(* IEC 61131-3 sources: std_i2980_v2.06_cp053/Source/IMM/ieccontrol/MoldHeightAdjust1 (part 4) *)

(* ---- ABButtonControl.pu ---- *)
IMPORT_OVER_LISTFILE
 IS_LINKED
, tyPanelButton
, tevPanelButtonRegisterData
, tevPanelButtonRegister
, ABManualButton
, tsDeviceId
, tsPanelButton

END_IMPORT

ALGORITHM_BLOCK ABButtonControl #DUMMY_EDIT_BLOCK

SYSTEM_VAR
 sv_bInitStart : BOOL;
 sv_bDeviceReady : BOOL;
 sv_iPanelMovementSelector : DINT;
 sv_bHMILedAutoAdjust_ledAttr : BYTE;
 sv_bHMILedAutoAdjust : BOOL;
 sv_PanelButtons : tyPanelButton;
 di_ButtonGeneral1 : BOOL;
 di_ButtonGeneral2 : BOOL;
 sv_DeviceId : tsDeviceId;
 di_ButtonStart : BOOL;
 sv_bButtonStart : BOOL;
END_VAR

SYSTEM_OBJECT
 evPanelButtonRegister : tevPanelButtonRegister;
 PU_Task_7 : TASK;
 PU_Task_13 : TASK;
END_OBJECT

VAR
 evPanelButtonRegisterData : tevPanelButtonRegisterData;
 abManualButton : ABManualButton;
 mpbButtonGeneralFwd : REFTO BOOL;
 mpbButtonGeneralBwd : REFTO BOOL;
 mbDIButtonStartLinked : BOOL;
 mbDIButtonGeneral1Linked : BOOL;
 mbDIButtonGeneral2Linked : BOOL;
 mpiPanelMovementSelector : REFTO DINT;
END_VAR

VAR CONSTANT
 cButtonMoveStart : DINT := 1;
END_VAR

POSTUPDATE_ALGORITHM pRegisterButtons ON PU_Task_13 WITH sv_bInitStart

#BEGIN_EDIT_BLOCK
(**************************************** WARNING ********************************************
 *** The KEBA Kemro K2 System including software is not intended for safety control tasks! ***
 ***                       For further information see Comment tab!                        ***
 *********************************************************************************************)

mpbButtonGeneralFwd := EMPTY;
mpbButtonGeneralBwd := EMPTY;

mbDIButtonStartLinked := IS_LINKED(di_ButtonStart);

mbDIButtonGeneral1Linked := IS_LINKED(di_ButtonGeneral1);
mbDIButtonGeneral2Linked := IS_LINKED(di_ButtonGeneral2);

IF (mbDIButtonGeneral1Linked AND mbDIButtonGeneral2Linked) THEN
    mpiPanelMovementSelector := @sv_iPanelMovementSelector;
END_IF;

// register start button
evPanelButtonRegisterData.Button.nPanelButtonType := nPanelButtonMovement;
evPanelButtonRegisterData.Button.iCompId := sv_DeviceId.CompId;
evPanelButtonRegisterData.Button.iIndexId := sv_DeviceId.IndexId;
evPanelButtonRegisterData.Button.iButtonId := cButtonMoveStart;
evPanelButtonRegisterData.Button.pbActionVar1 := @sv_bButtonStart;
evPanelButtonRegisterData.Button.pbActionVar2 := @sv_bButtonStart;
evPanelButtonRegisterData.Button.Optional.pbLedVar := @sv_bHMILedAutoAdjust;
evPanelButtonRegisterData.Button.Optional.piLedVarAttr := @sv_bHMILedAutoAdjust_ledAttr;
SET_EVENT(evPanelButtonRegister, evPanelButtonRegisterData);

;#END_EDIT_BLOCK END_ALGORITHM

POSTUPDATE_ALGORITHM pButtonStart ON PU_Task_7 WITH di_ButtonStart,sv_bButtonStart,mpbButtonGeneralBwd^,mpbButtonGeneralFwd^

VAR
 bButton : BOOL;
END_VAR
#BEGIN_EDIT_BLOCK
(**************************************** WARNING ********************************************
 *** The KEBA Kemro K2 System including software is not intended for safety control tasks! ***
 ***                       For further information see Comment tab!                        ***
 *********************************************************************************************)

// soft panel button
bButton := sv_bButtonStart;

// hw panel button
IF mbDIButtonStartLinked THEN
    bButton := bButton OR di_ButtonStart;
END_IF;

// external panel button
IF CHECK_REF(mpbButtonGeneralBwd^) THEN
    bButton := bButton OR mpbButtonGeneralBwd^;
END_IF;
IF CHECK_REF(mpbButtonGeneralFwd^) THEN
    bButton := bButton OR mpbButtonGeneralFwd^;
END_IF;

abManualButton.aButtonStart(bButtonStart := bButton);

;#END_EDIT_BLOCK END_ALGORITHM

POSTUPDATE_ALGORITHM pMoveSelectorChanged ON PU_Task_7 WITH mpiPanelMovementSelector^

VAR
 Button : tsPanelButton;
END_VAR
#BEGIN_EDIT_BLOCK
(**************************************** WARNING ********************************************
 *** The KEBA Kemro K2 System including software is not intended for safety control tasks! ***
 ***                       For further information see Comment tab!                        ***
 *********************************************************************************************)
mpbButtonGeneralFwd := EMPTY;
mpbButtonGeneralBwd := EMPTY;

IF (NOT sv_bDeviceReady) THEN
    // stop active movements
    abManualButton.aButtonStart(bButtonStart := FALSE);
END_IF;

IF (sv_iPanelMovementSelector > 0) THEN
    Button := sv_PanelButtons[sv_iPanelMovementSelector];
    IF (Button.iCompId = sv_DeviceId.CompId AND
        Button.iIndexId = sv_DeviceId.IndexId) THEN
        IF (Button.iButtonId = cButtonMoveStart) THEN
            mpbButtonGeneralFwd := @di_ButtonGeneral2;
            mpbButtonGeneralBwd := @di_ButtonGeneral1;
        END_IF;
    END_IF;
END_IF;

;#END_EDIT_BLOCK END_ALGORITHM

END_ALGORITHM_BLOCK

#END_OF_IEC_PART

@Puma @IecEditor 6 152 @Pou 25
@@@BEG_Comment@@@

@@@END_Comment@@@

@BEG_Contents

@BEG_Func
@RT(17)FuncTreeContainer
1
@Var @RT(9)IS_LINKED @RT(0) @T @T @DERIVED 0 @F @RT(22)KEBA_STANDARD_FUNCTION @F
@T
@BEG_Attrib
0 @RT(0) @RT(0)
@END_Attrib
1 1 @F @F @F @F

@END_Func

@BEG_Const
@RT(18)ConstTreeContainer
0
@END_Const

@BEG_Export

@BEG_Kind
@ALGORITHM_BLOCK @RT(15)ABButtonControl @STRUCTURED_TEXT
@RT(0) @RT(0) @RT(0)
@END_Kind

@BEG_Dcl
@RT(16)DclTreeContainer
23
@Var @RT(13)sv_bInitStart @RT(0) @T @T @RENAMED 0 @T @T @DT @RT(4)BOOL @RT(0) @T @T @BASIC 0 @F
@F @F
@T
@BEG_Attrib
3 @RT(0) @RT(0) @RT(0)
@END_Attrib
1 8 @F @F @F @F

@Var @RT(15)sv_bDeviceReady @RT(0) @T @T @RENAMED 0 @T @T @DT @RT(4)BOOL @RT(0) @T @T @BASIC 0 @F
@F @F
@T
@BEG_Attrib
3 @RT(0) @RT(0) @RT(0)
@END_Attrib
1 8 @F @F @F @F

@Var @RT(25)sv_iPanelMovementSelector @RT(0) @T @F @DT @RT(4)DINT @RT(0) @T @T @BASIC 0 @F
@F @F
@T
@BEG_Attrib
3 @RT(0) @RT(0) @RT(0)
@END_Attrib
1 8 @F @F @F @F

@Var @RT(28)sv_bHMILedAutoAdjust_ledAttr @RT(0) @T @F @DT @RT(4)BYTE @RT(0) @T @T @BASIC 0 @F
@F @F
@T
@BEG_Attrib
3 @RT(0) @RT(0) @RT(0)
@END_Attrib
1 8 @F @F @F @F

@Var @RT(20)sv_bHMILedAutoAdjust @RT(0) @T @F @DT @RT(4)BOOL @RT(0) @T @T @BASIC 0 @F
@F @F
@T
@BEG_Attrib
3 @RT(0) @RT(0) @RT(0)
@END_Attrib
1 8 @F @F @F @F

@Var @RT(15)sv_PanelButtons @RT(0) @T @T @DERIVED 0 @T @T @DT @RT(13)tyPanelButton @RT(0) @T @T @UNKNOWN 0 @F
@F @F
@T
@BEG_Attrib
3 @RT(0) @RT(0) @RT(0)
@END_Attrib
1 8 @F @F @F @F

@Var @RT(25)evPanelButtonRegisterData @RT(0) @T @T @DERIVED 0 @T @T @DT @RT(26)tevPanelButtonRegisterData @RT(0) @T @T @UNKNOWN 0 @F
@F @F
@T
@BEG_Attrib
3 @RT(0) @RT(0) @RT(0)
@END_Attrib
1 0 @F @F @F @F

@Var @RT(21)evPanelButtonRegister @RT(0) @T @T @DERIVED 0 @T @T @DT @RT(22)tevPanelButtonRegister @RT(0) @T @T @UNKNOWN 0 @F
@F @F
@T
@BEG_Attrib
3 @RT(0) @RT(0) @RT(0)
@END_Attrib
1 7 @F @F @F @F

@Var @RT(14)abManualButton @RT(0) @T @T @DERIVED 0 @T @T @DT @RT(14)ABManualButton @RT(0) @T @T @UNKNOWN 0 @F
@F @F
@T
@BEG_Attrib
3 @RT(0) @RT(0) @RT(0)
@END_Attrib
1 0 @F @F @F @F

@Var @RT(17)di_ButtonGeneral1 @RT(0) @T @F @DT @RT(4)BOOL @RT(0) @T @T @BASIC 0 @F
@F @F
@T
@BEG_Attrib
3 @RT(0) @RT(0) @RT(0)
@END_Attrib
1 8 @F @F @F @F

@Var @RT(17)di_ButtonGeneral2 @RT(0) @T @F @DT @RT(4)BOOL @RT(0) @T @T @BASIC 0 @F
@F @F
@T
@BEG_Attrib
3 @RT(0) @RT(0) @RT(0)
@END_Attrib
1 8 @F @F @F @F

@Var @RT(9)PU_Task_7 @RT(0) @T @F @DT @RT(4)TASK @RT(0) @T @T @BASIC 0 @F
@F @F
@T
@BEG_Attrib
3 @RT(0) @RT(0) @RT(0)
@END_Attrib
1 7 @F @F @F @F

@Var @RT(10)PU_Task_13 @RT(0) @T @T @RENAMED 0 @T @T @DT @RT(4)TASK @RT(0) @T @T @BASIC 0 @F
@F @F
@T
@BEG_Attrib
3 @RT(0) @RT(0) @RT(0)
@END_Attrib
1 7 @F @F @F @F

@Var @RT(11)sv_DeviceId @RT(0) @T @T @DERIVED 0 @T @T @DT @RT(10)tsDeviceId @RT(0) @T @T @UNKNOWN 0 @F
@F @F
@T
@BEG_Attrib
3 @RT(0) @RT(0) @RT(0)
@END_Attrib
1 8 @F @F @F @F

@Var @RT(16)cButtonMoveStart @RT(0) @T @F @DT @RT(4)DINT @RT(0) @T @T @BASIC 0 @F
@F @F
@T
@BEG_Attrib
3 @RT(1)1 @RT(0) @RT(0)
@END_Attrib
1 15 @F @F @F @F

@Var @RT(19)mpbButtonGeneralFwd @RT(0) @T @T @REFTO 0 @T @DT @RT(4)BOOL @RT(0) @T @T @BASIC 0 @F
@F @F
@T
@BEG_Attrib
3 @RT(0) @RT(0) @RT(0)
@END_Attrib
1 0 @F @F @F @F

@Var @RT(19)mpbButtonGeneralBwd @RT(0) @T @T @REFTO 0 @T @DT @RT(4)BOOL @RT(0) @T @T @BASIC 0 @F
@F @F
@T
@BEG_Attrib
3 @RT(0) @RT(0) @RT(0)
@END_Attrib
1 0 @F @F @F @F

@Var @RT(21)mbDIButtonStartLinked @RT(0) @T @F @DT @RT(4)BOOL @RT(0) @T @T @BASIC 0 @F
@F @F
@T
@BEG_Attrib
3 @RT(0) @RT(0) @RT(0)
@END_Attrib
1 0 @F @F @F @F

@Var @RT(24)mbDIButtonGeneral1Linked @RT(0) @T @F @DT @RT(4)BOOL @RT(0) @T @T @BASIC 0 @F
@F @F
@T
@BEG_Attrib
3 @RT(0) @RT(0) @RT(0)
@END_Attrib
1 0 @F @F @F @F

@Var @RT(24)mbDIButtonGeneral2Linked @RT(0) @T @F @DT @RT(4)BOOL @RT(0) @T @T @BASIC 0 @F
@F @F
@T
@BEG_Attrib
3 @RT(0) @RT(0) @RT(0)
@END_Attrib
1 0 @F @F @F @F

@Var @RT(14)di_ButtonStart @RT(0) @T @T @RENAMED 0 @T @T @DT @RT(4)BOOL @RT(0) @T @T @BASIC 0 @F
@F @F
@T
@BEG_Attrib
3 @RT(0) @RT(0) @RT(0)
@END_Attrib
1 8 @F @F @F @F

@Var @RT(15)sv_bButtonStart @RT(0) @T @T @RENAMED 0 @T @T @DT @RT(4)BOOL @RT(0) @T @T @BASIC 0 @F
@F @F
@T
@BEG_Attrib
3 @RT(0) @RT(0) @RT(0)
@END_Attrib
1 8 @F @F @F @F

@Var @RT(24)mpiPanelMovementSelector @RT(0) @T @T @REFTO 0 @T @DT @RT(4)DINT @RT(0) @T @T @BASIC 0 @F
@F @F
@T
@BEG_Attrib
3 @RT(0) @RT(0) @RT(0)
@END_Attrib
1 0 @F @F @F @F

@END_Dcl

@END_Export

@BEG_Body

3

@BEG_Export

@BEG_Algo
@POSTUPDATE_ALGORITHM @RT(16)pRegisterButtons @STRUCTURED_TEXT
@RT(0) @RT(13)sv_bInitStart @RT(10)PU_Task_13 @F @F
@END_Algo

@BEG_Dcl
@RT(16)DclTreeContainer
0
@END_Dcl

@END_Export

@BEG_Export

@BEG_Algo
@POSTUPDATE_ALGORITHM @RT(12)pButtonStart @STRUCTURED_TEXT
@RT(0) @RT(72)di_ButtonStart,sv_bButtonStart,mpbButtonGeneralBwd^,mpbButtonGeneralFwd^ @RT(9)PU_Task_7 @F @F
@END_Algo

@BEG_Dcl
@RT(16)DclTreeContainer
1
@Var @RT(7)bButton @RT(0) @T @F @DT @RT(4)BOOL @RT(0) @T @T @BASIC 0 @F
@F @F
@T
@BEG_Attrib
3 @RT(0) @RT(0) @RT(0)
@END_Attrib
1 0 @F @F @F @F

@END_Dcl

@END_Export

@BEG_Export

@BEG_Algo
@POSTUPDATE_ALGORITHM @RT(20)pMoveSelectorChanged @STRUCTURED_TEXT
@RT(0) @RT(25)mpiPanelMovementSelector^ @RT(9)PU_Task_7 @F @F
@END_Algo

@BEG_Dcl
@RT(16)DclTreeContainer
1
@Var @RT(6)Button @RT(0) @T @T @DERIVED 0 @T @T @DT @RT(13)tsPanelButton @RT(0) @T @T @UNKNOWN 0 @F
@F @F
@T
@BEG_Attrib
3 @RT(0) @RT(0) @RT(0)
@END_Attrib
1 0 @F @F @F @F

@END_Dcl

@END_Export

@BEG_Body
@TL(29)
(**************************************** WARNING ********************************************
 *** The KEBA Kemro K2 System including software is not intended for safety control tasks! ***
 ***                       For further information see Comment tab!                        ***
 *********************************************************************************************)

mpbButtonGeneralFwd := EMPTY;
mpbButtonGeneralBwd := EMPTY;

mbDIButtonStartLinked := IS_LINKED(di_ButtonStart);

mbDIButtonGeneral1Linked := IS_LINKED(di_ButtonGeneral1);
mbDIButtonGeneral2Linked := IS_LINKED(di_ButtonGeneral2);

IF (mbDIButtonGeneral1Linked AND mbDIButtonGeneral2Linked) THEN
    mpiPanelMovementSelector := @sv_iPanelMovementSelector;
END_IF;

// register start button
evPanelButtonRegisterData.Button.nPanelButtonType := nPanelButtonMovement;
evPanelButtonRegisterData.Button.iCompId := sv_DeviceId.CompId;
evPanelButtonRegisterData.Button.iIndexId := sv_DeviceId.IndexId;
evPanelButtonRegisterData.Button.iButtonId := cButtonMoveStart;
evPanelButtonRegisterData.Button.pbActionVar1 := @sv_bButtonStart;
evPanelButtonRegisterData.Button.pbActionVar2 := @sv_bButtonStart;
evPanelButtonRegisterData.Button.Optional.pbLedVar := @sv_bHMILedAutoAdjust;
evPanelButtonRegisterData.Button.Optional.piLedVarAttr := @sv_bHMILedAutoAdjust_ledAttr;
SET_EVENT(evPanelButtonRegister, evPanelButtonRegisterData);

@END_Body

@@@BEG_Comment@@@
@TL(0)

@@@END_Comment@@@

@BEG_Body
@TL(24)
(**************************************** WARNING ********************************************
 *** The KEBA Kemro K2 System including software is not intended for safety control tasks! ***
 ***                       For further information see Comment tab!                        ***
 *********************************************************************************************)

// soft panel button
bButton := sv_bButtonStart;

// hw panel button
IF mbDIButtonStartLinked THEN
    bButton := bButton OR di_ButtonStart;
END_IF;

// external panel button
IF CHECK_REF(mpbButtonGeneralBwd^) THEN
    bButton := bButton OR mpbButtonGeneralBwd^;
END_IF;
IF CHECK_REF(mpbButtonGeneralFwd^) THEN
    bButton := bButton OR mpbButtonGeneralFwd^;
END_IF;

abManualButton.aButtonStart(bButtonStart := bButton);

@END_Body

@@@BEG_Comment@@@
@TL(0)

@@@END_Comment@@@

@BEG_Body
@TL(26)
(**************************************** WARNING ********************************************
 *** The KEBA Kemro K2 System including software is not intended for safety control tasks! ***
 ***                       For further information see Comment tab!                        ***
 *********************************************************************************************)
mpbButtonGeneralFwd := EMPTY;
mpbButtonGeneralBwd := EMPTY;

IF (NOT sv_bDeviceReady) THEN
    // stop active movements
    abManualButton.aButtonStart(bButtonStart := FALSE);
END_IF;

IF (sv_iPanelMovementSelector > 0) THEN
    Button := sv_PanelButtons[sv_iPanelMovementSelector];
    IF (Button.iCompId = sv_DeviceId.CompId AND
        Button.iIndexId = sv_DeviceId.IndexId) THEN
        IF (Button.iButtonId = cButtonMoveStart) THEN
            mpbButtonGeneralFwd := @di_ButtonGeneral2;
            mpbButtonGeneralBwd := @di_ButtonGeneral1;
        END_IF;
    END_IF;
END_IF;

@END_Body

@@@BEG_Comment@@@
@TL(0)

@@@END_Comment@@@
@END_Body

@END_Contents

(* ---- ABCalculateMoldHeightImpulses.pu ---- *)
(*
Calculate number of mold height adjust impulses from clamp force
and clamp force from mold height adjust impulses
*)

IMPORT_OVER_LISTFILE
 KCTRL_Lintab_Light
, KAPPL_LintabData
, KCTRL_Lintab_Param_Light

END_IMPORT

ALGORITHM_BLOCK ABCalculateMoldHeightImpulses #DUMMY_EDIT_BLOCK

VAR
 abKCTRL_Lintab : KCTRL_Lintab_Light;
END_VAR

ALGORITHM aInit

VAR_INPUT
 Lintab : KAPPL_LintabData (* lintab for calculating number of impulses from clamping force *);
END_VAR

VAR_TEMP
 LintabParam : KCTRL_Lintab_Param_Light;
END_VAR
#BEGIN_EDIT_BLOCK
(**************************************** WARNING ********************************************
 *** The KEBA Kemro K2 System including software is not intended for safety control tasks! ***
 ***                       For further information see Comment tab!                        ***
 *********************************************************************************************)

LintabParam.LintabPoints := Lintab.LintabPoints;
LintabParam.Mode.bLinearExtrapolation := TRUE;
LintabParam.Mode.bSetNegativeValuesToZero := TRUE;
LintabParam.Mode.bZeroExtrapolation := FALSE;
abKCTRL_Lintab.Par(Param := LintabParam);
abKCTRL_Lintab.Init();

;#END_EDIT_BLOCK END_ALGORITHM

ALGORITHM aCalc

VAR_INPUT
 rForce : REAL (* wanted clamping force *);
END_VAR

VAR_OUTPUT
 iImpulses : DINT (* number of impulses needed for given force *);
END_VAR
#BEGIN_EDIT_BLOCK
(**************************************** WARNING ********************************************
 *** The KEBA Kemro K2 System including software is not intended for safety control tasks! ***
 ***                       For further information see Comment tab!                        ***
 *********************************************************************************************)

//calculate number of impulses from clamping force lintab

abKCTRL_Lintab.CalculateInv(rY := rForce);
iImpulses := REAL_TO_DINT(abKCTRL_Lintab.CalculateInv.rX);

;#END_EDIT_BLOCK END_ALGORITHM

ALGORITHM aCalcInv

VAR_INPUT
 iImpulses : DINT (* number of impulses *);
END_VAR

VAR_OUTPUT
 rForce : REAL (* force from given number of impulses *);
END_VAR
#BEGIN_EDIT_BLOCK
(**************************************** WARNING ********************************************
 *** The KEBA Kemro K2 System including software is not intended for safety control tasks! ***
 ***                       For further information see Comment tab!                        ***
 *********************************************************************************************)

abKCTRL_Lintab.Calculate(rX := DINT_TO_REAL(iImpulses));
rForce := abKCTRL_Lintab.Calculate.rY;

;#END_EDIT_BLOCK END_ALGORITHM

END_ALGORITHM_BLOCK

#END_OF_IEC_PART

@Puma @IecEditor 6 30 @Pou 25
@@@BEG_Comment@@@
Calculate number of mold height adjust impulses from clamp force
and clamp force from mold height adjust impulses
@@@END_Comment@@@

@BEG_Contents

@BEG_Func
@RT(17)FuncTreeContainer
0
@END_Func

@BEG_Const
@RT(18)ConstTreeContainer
0
@END_Const

@BEG_Export

@BEG_Kind
@ALGORITHM_BLOCK @RT(29)ABCalculateMoldHeightImpulses @STRUCTURED_TEXT
@RT(0) @RT(0) @RT(0)
@END_Kind

@BEG_Dcl
@RT(16)DclTreeContainer
1
@Var @RT(14)abKCTRL_Lintab @RT(0) @T @T @DERIVED 0 @T @T @DT @RT(18)KCTRL_Lintab_Light @RT(0) @T @T @UNKNOWN 0 @F
@F @F
@T
@BEG_Attrib
3 @RT(0) @RT(0) @RT(0)
@END_Attrib
1 0 @F @F @F @F

@END_Dcl

@END_Export

@BEG_Body

3

@BEG_Export

@BEG_Algo
@ALGORITHM @RT(5)aInit @STRUCTURED_TEXT
@RT(0) @RT(0) @RT(0) @F @F
@END_Algo

@BEG_Dcl
@RT(16)DclTreeContainer
2
@Var @RT(6)Lintab @RT(0) @T @T @DERIVED 0 @T @T @DT @RT(16)KAPPL_LintabData @RT(0) @T @T @UNKNOWN 0 @F
@F @F
@T
@BEG_Attrib
3 @RT(0) @RT(61)lintab for calculating number of impulses from clamping force @RT(0)
@END_Attrib
1 1 @F @F @F @F

@Var @RT(11)LintabParam @RT(0) @T @T @DERIVED 0 @T @T @DT @RT(24)KCTRL_Lintab_Param_Light @RT(0) @T @T @UNKNOWN 0 @F
@F @F
@T
@BEG_Attrib
3 @RT(0) @RT(0) @RT(0)
@END_Attrib
1 4 @F @F @F @F

@END_Dcl

@END_Export

@BEG_Export

@BEG_Algo
@ALGORITHM @RT(5)aCalc @STRUCTURED_TEXT
@RT(0) @RT(0) @RT(0) @F @F
@END_Algo

@BEG_Dcl
@RT(16)DclTreeContainer
2
@Var @RT(6)rForce @RT(0) @T @F @DT @RT(4)REAL @RT(0) @T @T @BASIC 0 @F
@F @F
@T
@BEG_Attrib
3 @RT(0) @RT(21)wanted clamping force @RT(0)
@END_Attrib
1 1 @F @F @F @F

@Var @RT(9)iImpulses @RT(0) @T @F @DT @RT(4)DINT @RT(0) @T @T @BASIC 0 @F
@F @F
@T
@BEG_Attrib
3 @RT(0) @RT(41)number of impulses needed for given force @RT(0)
@END_Attrib
1 3 @F @F @F @F

@END_Dcl

@END_Export

@BEG_Export

@BEG_Algo
@ALGORITHM @RT(8)aCalcInv @STRUCTURED_TEXT
@RT(0) @RT(0) @RT(0) @F @F
@END_Algo

@BEG_Dcl
@RT(16)DclTreeContainer
2
@Var @RT(9)iImpulses @RT(0) @T @F @DT @RT(4)DINT @RT(0) @T @T @BASIC 0 @F
@F @F
@T
@BEG_Attrib
3 @RT(0) @RT(18)number of impulses @RT(0)
@END_Attrib
1 1 @F @F @F @F

@Var @RT(6)rForce @RT(0) @T @F @DT @RT(4)REAL @RT(0) @T @T @BASIC 0 @F
@F @F
@T
@BEG_Attrib
3 @RT(0) @RT(35)force from given number of impulses @RT(0)
@END_Attrib
1 3 @F @F @F @F

@END_Dcl

@END_Export

@BEG_Body
@TL(12)
(**************************************** WARNING ********************************************
 *** The KEBA Kemro K2 System including software is not intended for safety control tasks! ***
 ***                       For further information see Comment tab!                        ***
 *********************************************************************************************)

LintabParam.LintabPoints := Lintab.LintabPoints;
LintabParam.Mode.bLinearExtrapolation := TRUE;
LintabParam.Mode.bSetNegativeValuesToZero := TRUE;
LintabParam.Mode.bZeroExtrapolation := FALSE;
abKCTRL_Lintab.Par(Param := LintabParam);
abKCTRL_Lintab.Init();

@END_Body

@@@BEG_Comment@@@
@TL(0)

@@@END_Comment@@@

@BEG_Body
@TL(11)
(**************************************** WARNING ********************************************
 *** The KEBA Kemro K2 System including software is not intended for safety control tasks! ***
 ***                       For further information see Comment tab!                        ***
 *********************************************************************************************)

//calculate number of impulses from clamping force lintab

abKCTRL_Lintab.CalculateInv(rY := rForce);
iImpulses := REAL_TO_DINT(abKCTRL_Lintab.CalculateInv.rX);

@END_Body

@@@BEG_Comment@@@
@TL(0)

@@@END_Comment@@@

@BEG_Body
@TL(9)
(**************************************** WARNING ********************************************
 *** The KEBA Kemro K2 System including software is not intended for safety control tasks! ***
 ***                       For further information see Comment tab!                        ***
 *********************************************************************************************)

abKCTRL_Lintab.Calculate(rX := DINT_TO_REAL(iImpulses));
rForce := abKCTRL_Lintab.Calculate.rY;

@END_Body

@@@BEG_Comment@@@
@TL(0)

@@@END_Comment@@@
@END_Body

@END_Contents

(* ---- ABCalculateMoldHeightMm.pu ---- *)
(*
Calculate number of mold height adjust impulses from clamp force
and clamp force from mold height adjust impulses
*)

IMPORT_OVER_LISTFILE
 KCTRL_Lintab_Light
, KAPPL_LintabData
, KCTRL_Lintab_Param_Light

END_IMPORT

ALGORITHM_BLOCK ABCalculateMoldHeightMm #DUMMY_EDIT_BLOCK

VAR
 abKCTRL_Lintab_ClampF : KCTRL_Lintab_Light;
 abKCTRL_Lintab_ToggleLever : KCTRL_Lintab_Light;
END_VAR

ALGORITHM aInit

VAR_INPUT
 LintabClampF : KAPPL_LintabData (* lintab for calculating mold open length from clamping force *);
 LintabToggleLever : KAPPL_LintabData (* lintab for calculating mold open length from clamping force *);
END_VAR

VAR_TEMP
 LintabParam : KCTRL_Lintab_Param_Light;
END_VAR
#BEGIN_EDIT_BLOCK
(**************************************** WARNING ********************************************
 *** The KEBA Kemro K2 System including software is not intended for safety control tasks! ***
 ***                       For further information see Comment tab!                        ***
 *********************************************************************************************)

LintabParam.Mode.bLinearExtrapolation := TRUE;
LintabParam.Mode.bSetNegativeValuesToZero := TRUE;
LintabParam.Mode.bZeroExtrapolation := FALSE;

LintabParam.LintabPoints := LintabClampF.LintabPoints;
abKCTRL_Lintab_ClampF.Par(Param := LintabParam);
abKCTRL_Lintab_ClampF.Init();

LintabParam.LintabPoints := LintabToggleLever.LintabPoints;
abKCTRL_Lintab_ToggleLever.Par(Param := LintabParam);
abKCTRL_Lintab_ToggleLever.Init();

;#END_EDIT_BLOCK END_ALGORITHM

ALGORITHM aCalc

VAR_INPUT
 rForce : REAL (* wanted clamping force *);
END_VAR

VAR_OUTPUT
 rToggleLeverPos : REAL (* new mold offset for given force *);
 rMoldPos : REAL;
END_VAR
#BEGIN_EDIT_BLOCK
(**************************************** WARNING ********************************************
 *** The KEBA Kemro K2 System including software is not intended for safety control tasks! ***
 ***                       For further information see Comment tab!                        ***
 *********************************************************************************************)

//length mold has to open from clamping force lintab

abKCTRL_Lintab_ClampF.CalculateInv(rY := rForce);
rMoldPos := abKCTRL_Lintab_ClampF.CalculateInv.rX;

//getting eqivalent toggleleverpos
abKCTRL_Lintab_ToggleLever.CalculateInv(rY := rMoldPos);
rToggleLeverPos := abKCTRL_Lintab_ToggleLever.CalculateInv.rX;

;#END_EDIT_BLOCK END_ALGORITHM

ALGORITHM aCalcInv

// VAR_INPUT
 // rMoldPos : REAL (* mold position *);
// END_VAR

// VAR_OUTPUT
 // rForce : REAL (* force from given number of impulses *);
// END_VAR
#BEGIN_EDIT_BLOCK
(**************************************** WARNING ********************************************
 *** The KEBA Kemro K2 System including software is not intended for safety control tasks! ***
 ***                       For further information see Comment tab!                        ***
 *********************************************************************************************)

//abKCTRL_Lintab.Calculate(rX := rMoldPos);
//rForce := abKCTRL_Lintab.Calculate.rY;

;#END_EDIT_BLOCK END_ALGORITHM

END_ALGORITHM_BLOCK

#END_OF_IEC_PART

@Puma @IecEditor 6 68 @Pou 25
@@@BEG_Comment@@@
Calculate number of mold height adjust impulses from clamp force
and clamp force from mold height adjust impulses
@@@END_Comment@@@

@BEG_Contents

@BEG_Func
@RT(17)FuncTreeContainer
0
@END_Func

@BEG_Const
@RT(18)ConstTreeContainer
0
@END_Const

@BEG_Export

@BEG_Kind
@ALGORITHM_BLOCK @RT(23)ABCalculateMoldHeightMm @STRUCTURED_TEXT
@RT(0) @RT(0) @RT(0)
@END_Kind

@BEG_Dcl
@RT(16)DclTreeContainer
2
@Var @RT(21)abKCTRL_Lintab_ClampF @RT(0) @T @T @DERIVED 0 @T @T @DT @RT(18)KCTRL_Lintab_Light @RT(0) @T @T @UNKNOWN 0 @F
@F @F
@T
@BEG_Attrib
3 @RT(0) @RT(0) @RT(0)
@END_Attrib
1 0 @F @F @F @F

@Var @RT(26)abKCTRL_Lintab_ToggleLever @RT(0) @T @T @DERIVED 0 @T @T @DT @RT(18)KCTRL_Lintab_Light @RT(0) @T @T @UNKNOWN 0 @F
@F @F
@T
@BEG_Attrib
3 @RT(0) @RT(0) @RT(0)
@END_Attrib
1 0 @F @F @F @F

@END_Dcl

@END_Export

@BEG_Body

3

@BEG_Export

@BEG_Algo
@ALGORITHM @RT(5)aInit @STRUCTURED_TEXT
@RT(0) @RT(0) @RT(0) @F @F
@END_Algo

@BEG_Dcl
@RT(16)DclTreeContainer
3
@Var @RT(12)LintabClampF @RT(0) @T @T @DERIVED 0 @T @T @DT @RT(16)KAPPL_LintabData @RT(0) @T @T @UNKNOWN 0 @F
@F @F
@T
@BEG_Attrib
3 @RT(0) @RT(59)lintab for calculating mold open length from clamping force @RT(0)
@END_Attrib
1 1 @F @F @F @F

@Var @RT(17)LintabToggleLever @RT(0) @T @T @DERIVED 0 @T @T @DT @RT(16)KAPPL_LintabData @RT(0) @T @T @UNKNOWN 0 @F
@F @F
@T
@BEG_Attrib
3 @RT(0) @RT(59)lintab for calculating mold open length from clamping force @RT(0)
@END_Attrib
1 1 @F @F @F @F

@Var @RT(11)LintabParam @RT(0) @T @T @DERIVED 0 @T @T @DT @RT(24)KCTRL_Lintab_Param_Light @RT(0) @T @T @UNKNOWN 0 @F
@F @F
@T
@BEG_Attrib
3 @RT(0) @RT(0) @RT(0)
@END_Attrib
1 4 @F @F @F @F

@END_Dcl

@END_Export

@BEG_Export

@BEG_Algo
@ALGORITHM @RT(5)aCalc @STRUCTURED_TEXT
@RT(0) @RT(0) @RT(0) @F @F
@END_Algo

@BEG_Dcl
@RT(16)DclTreeContainer
3
@Var @RT(6)rForce @RT(0) @T @F @DT @RT(4)REAL @RT(0) @T @T @BASIC 0 @F
@F @F
@T
@BEG_Attrib
3 @RT(0) @RT(21)wanted clamping force @RT(0)
@END_Attrib
1 1 @F @F @F @F

@Var @RT(15)rToggleLeverPos @RT(0) @T @F @DT @RT(4)REAL @RT(0) @T @T @BASIC 0 @F
@F @F
@T
@BEG_Attrib
3 @RT(0) @RT(31)new mold offset for given force @RT(0)
@END_Attrib
1 3 @F @F @F @F

@Var @RT(8)rMoldPos @RT(0) @T @F @DT @RT(4)REAL @RT(0) @T @T @BASIC 0 @F
@F @F
@T
@BEG_Attrib
3 @RT(0) @RT(0) @RT(0)
@END_Attrib
1 3 @F @F @F @F

@END_Dcl

@END_Export

@BEG_Export

@BEG_Algo
@ALGORITHM @RT(8)aCalcInv @STRUCTURED_TEXT
@RT(0) @RT(0) @RT(0) @F @F
@END_Algo

@BEG_Dcl
@RT(16)DclTreeContainer
2
@Var @RT(8)rMoldPos @RT(0) @T @F @DT @RT(4)REAL @RT(0) @T @T @BASIC 0 @F
@F @T
@T
@BEG_Attrib
3 @RT(0) @RT(13)mold position @RT(0)
@END_Attrib
1 1 @F @F @F @F

@Var @RT(6)rForce @RT(0) @T @F @DT @RT(4)REAL @RT(0) @T @T @BASIC 0 @F
@F @T
@T
@BEG_Attrib
3 @RT(0) @RT(35)force from given number of impulses @RT(0)
@END_Attrib
1 3 @F @F @F @F

@END_Dcl

@END_Export

@BEG_Body
@TL(18)
(**************************************** WARNING ********************************************
 *** The KEBA Kemro K2 System including software is not intended for safety control tasks! ***
 ***                       For further information see Comment tab!                        ***
 *********************************************************************************************)

LintabParam.Mode.bLinearExtrapolation := TRUE;
LintabParam.Mode.bSetNegativeValuesToZero := TRUE;
LintabParam.Mode.bZeroExtrapolation := FALSE;

LintabParam.LintabPoints := LintabClampF.LintabPoints;
abKCTRL_Lintab_ClampF.Par(Param := LintabParam);
abKCTRL_Lintab_ClampF.Init();

LintabParam.LintabPoints := LintabToggleLever.LintabPoints;
abKCTRL_Lintab_ToggleLever.Par(Param := LintabParam);
abKCTRL_Lintab_ToggleLever.Init();

@END_Body

@@@BEG_Comment@@@
@TL(0)

@@@END_Comment@@@

@BEG_Body
@TL(16)
(**************************************** WARNING ********************************************
 *** The KEBA Kemro K2 System including software is not intended for safety control tasks! ***
 ***                       For further information see Comment tab!                        ***
 *********************************************************************************************)

//length mold has to open from clamping force lintab

abKCTRL_Lintab_ClampF.CalculateInv(rY := rForce);
rMoldPos := abKCTRL_Lintab_ClampF.CalculateInv.rX;

//getting eqivalent toggleleverpos
abKCTRL_Lintab_ToggleLever.CalculateInv(rY := rMoldPos);
rToggleLeverPos := abKCTRL_Lintab_ToggleLever.CalculateInv.rX;

@END_Body

@@@BEG_Comment@@@
@TL(0)

@@@END_Comment@@@

@BEG_Body
@TL(9)
(**************************************** WARNING ********************************************
 *** The KEBA Kemro K2 System including software is not intended for safety control tasks! ***
 ***                       For further information see Comment tab!                        ***
 *********************************************************************************************)

//abKCTRL_Lintab.Calculate(rX := rMoldPos);
//rForce := abKCTRL_Lintab.Calculate.rY;

@END_Body

@@@BEG_Comment@@@
@TL(0)

@@@END_Comment@@@
@END_Body

@END_Contents

(* ---- ABManualButton.pu ---- *)
(*
@h    ! WARNING !
@h    The Kemro K2 system (including software) only meets category B according to EN 954-1,
@h    thus it is not intended for usage in safety-relevant control applications in the field
@h    of personal safety (e.g. emergency stop).
@h    To implement potentially necessary safety-relevant control tasks, always use additional
@h    external safety devices that are intended for the particular purpose, and meet the necessary
@h    functional safety.
@h    For further information see EN 954-1 (EN ISO 13849-1) and/or the K2-x00 user manual, chapter
@h    "CE conformity, directives and standards".

This algo block starts the automatic mold height adjustment by calling the
system.FBManualButton with the correct parameters corresponding to a pressed Panel Button.
*)

IMPORT_OVER_LISTFILE
 SET_ALARM
, nSetup
, cCompMold
, cCompMoldHeight
, tevStartedStopped
, tsMoveData
, tnOperationMode
, tsDeviceId
, FBManualButtonKeep
, tsAlarm
, FBCheckReady
, FBCheckPosReached
, tevStartedStoppedData

END_IMPORT

ALGORITHM_BLOCK ABManualButton #DUMMY_EDIT_BLOCK

SYSTEM_VAR
 sv_MoveMoldHeightAuto : tsMoveData;
 sv_bAutoMoldHeightAdjustActive : BOOL (* is TRUE when auto mold height adjust is acitve *);
 sv_bLedAutoAdjust_ledAttr : BYTE (* LED Attribute *);
 sv_bHMILedAutoAdjust : BOOL;
 sv_bHMILedAutoAdjust_ledAttr : BYTE (* LED Attribute *);
 sv_bLedAutoAdjust : BOOL;
 sv_bInitStart : BOOL;
 sv_OperationMode : tnOperationMode;
 sv_bInitDone : BOOL;
 sv_DeviceId : tsDeviceId;
 sv_bMoldHeightAutoAdjHMI : BOOL (* hmi can start/stop automh adjust with this SV *);
 sv_bDeviceReady : BOOL;
END_VAR

SYSTEM_OBJECT
 PU_Task_7 : TASK;
 EV_Task_7 : TASK;
 erSetupModeRequiredForAdjust : ALARM;
 evStartedStopped : tevStartedStopped;
END_OBJECT

VAR_EXTERNAL
 g_b2Platen : BOOL;
END_VAR

VAR
 fbManualButton : FBManualButtonKeep;
 mpbMoldReady : REFTO BOOL;
 mpbMoldHeightReady : REFTO BOOL;
 mpbNutsOpen : REFTO BOOL;
 mAlarmNutsNotOpen : tsAlarm;
END_VAR

(*
This algo starts the mold height automatic adjustment by calling the
system.FBManualButton with the correct parameters when the di_ButtonIn is
pressed. (post update).
*)

ALGORITHM aStartStop

VAR_INPUT
 bStart : BOOL;
END_VAR
#BEGIN_EDIT_BLOCK
(**************************************** WARNING ********************************************
 *** The KEBA Kemro K2 System including software is not intended for safety control tasks! ***
 ***                       For further information see Comment tab!                        ***
 *********************************************************************************************)

IF (bStart AND (sv_OperationMode <> nSetup)) THEN
   //ignore button if operation mode is not setup
   SET_ALARM(Name := erSetupModeRequiredForAdjust,
            SubID1 := sv_DeviceId.CompId);
   sv_bMoldHeightAutoAdjHMI := FALSE;
   RETURN;
END_IF;

IF bStart AND g_b2Platen THEN
   //ignore button if lock nuts are not open
   IF NOT mpbNutsOpen^ THEN
      SET_ALARM(Name := mAlarmNutsNotOpen.AlarmId);
      sv_bMoldHeightAutoAdjHMI := FALSE;
      RETURN;
   END_IF;
END_IF;

IF (bStart AND sv_bDeviceReady) THEN
   IF (mpbMoldReady <> EMPTY AND NOT mpbMoldReady^) OR (mpbMoldHeightReady <> EMPTY AND NOT mpbMoldHeightReady^) THEN
      // auto adjust should be started and mold movement or mold adjust movement acitve
      // -> ignore manual button
      RETURN;
   END_IF;
END_IF;

(*@ MoldHeightAdjustN.ABManualButton.pButtonStart.Call the fbManualButton using the sv_MoveMoldHeightAuto parameters *)
IF (bStart AND sv_bDeviceReady) OR ((NOT bStart) AND (NOT sv_bDeviceReady)) THEN
   fbManualButton(bButton := TRUE, MoveId := sv_MoveMoldHeightAuto.MoveId, MoveDir := sv_MoveMoldHeightAuto.MoveDir);
END_IF;

;#END_EDIT_BLOCK END_ALGORITHM

(*
This algo starts the mold height automatic adjustment by calling the
system.FBManualButton with the correct parameters when the di_ButtonIn is
pressed. (post update).
*)

ALGORITHM aButtonStart

VAR_INPUT
 bButtonStart : BOOL;
END_VAR
#BEGIN_EDIT_BLOCK
(**************************************** WARNING ********************************************
 *** The KEBA Kemro K2 System including software is not intended for safety control tasks! ***
 ***                       For further information see Comment tab!                        ***
 *********************************************************************************************)

IF bButtonStart THEN
    sv_bMoldHeightAutoAdjHMI := NOT sv_bMoldHeightAutoAdjHMI;
END_IF;

;#END_EDIT_BLOCK END_ALGORITHM

(*
This algo starts the mold height automatic adjustment by calling the
system.FBManualButton with the correct parameters when the di_ButtonIn is
pressed. (post update).
*)

POSTUPDATE_ALGORITHM pHMIStart ON PU_Task_7 WITH sv_bMoldHeightAutoAdjHMI

#BEGIN_EDIT_BLOCK
(**************************************** WARNING ********************************************
 *** The KEBA Kemro K2 System including software is not intended for safety control tasks! ***
 ***                       For further information see Comment tab!                        ***
 *********************************************************************************************)

IF (sv_bMoldHeightAutoAdjHMI AND sv_bDeviceReady) THEN
    aStartStop(TRUE);
ELSIF ((NOT sv_bMoldHeightAutoAdjHMI) AND (NOT sv_bDeviceReady)) THEN
    aStartStop(FALSE);
END_IF;

;#END_EDIT_BLOCK END_ALGORITHM

POSTUPDATE_ALGORITHM pLedControl ON PU_Task_7 WITH sv_bAutoMoldHeightAdjustActive,sv_bInitStart

VAR
 bInitDone : BOOL;
 mbLedAutoAdjustExists : BOOL := FALSE;
END_VAR
#BEGIN_EDIT_BLOCK
(**************************************** WARNING ********************************************
 *** The KEBA Kemro K2 System including software is not intended for safety control tasks! ***
 ***                       For further information see Comment tab!                        ***
 *********************************************************************************************)

IF NOT bInitDone THEN
    sv_bHMILedAutoAdjust_ledAttr := 16#3;
    IF IS_LINKED(sv_bLedAutoAdjust) AND IS_LINKED(sv_bLedAutoAdjust_ledAttr) THEN
        sv_bLedAutoAdjust_ledAttr := sv_bHMILedAutoAdjust_ledAttr;
        mbLedAutoAdjustExists := TRUE;
    ELSE
        mbLedAutoAdjustExists := FALSE;
    END_IF;

    bInitDone := TRUE;
END_IF;

sv_bHMILedAutoAdjust := sv_bAutoMoldHeightAdjustActive;
IF mbLedAutoAdjustExists THEN
    sv_bLedAutoAdjust := sv_bHMILedAutoAdjust;
END_IF;

;#END_EDIT_BLOCK END_ALGORITHM

POSTUPDATE_ALGORITHM pInitDone ON PU_Task_7(10) WITH sv_bInitDone

VAR
 fbCheckReady : FBCheckReady;
 DeviceId : tsDeviceId;
 fbCheckPosReached : FBCheckPosReached;
END_VAR
#BEGIN_EDIT_BLOCK
(**************************************** WARNING ********************************************
 *** The KEBA Kemro K2 System including software is not intended for safety control tasks! ***
 ***                       For further information see Comment tab!                        ***
 *********************************************************************************************)

//get reference to ready flag of mold function unit
DeviceId.CompId := cCompMold;
DeviceId.IndexId := sv_DeviceId.IndexId;
fbCheckReady(DeviceId := DeviceId);
mpbMoldReady := fbCheckReady.pbReady;

//get reference to ready flag of mold adjust function unit
DeviceId.CompId := cCompMoldHeight;
DeviceId.IndexId := sv_DeviceId.IndexId;
fbCheckReady(DeviceId := DeviceId);
mpbMoldHeightReady := fbCheckReady.pbReady;

//get reference to mold nut open movement and save according alarm
IF g_b2Platen THEN
   DeviceId.CompId := cCompMoldNuts;
   DeviceId.IndexId := sv_DeviceId.IndexId;
   fbCheckPosReached(DeviceId := DeviceId,
                     MoveDir := cMoveOpen,
                     MoveId := cMoveOpen);

   mpbNutsOpen := fbCheckPosReached.pbPosReached;
   mAlarmNutsNotOpen := fbCheckPosReached.Alarm;
END_IF;

;#END_EDIT_BLOCK END_ALGORITHM

(*
Manage list and count of currently started movments
in sv_StartedMovements when receiving evStartedStopped events
*)

EVENT_ALGORITHM evaStartedStopped ON EV_Task_7 WITH evStartedStopped

VAR_INPUT
 evStartedStoppedData : tevStartedStoppedData;
END_VAR
#BEGIN_EDIT_BLOCK
(**************************************** WARNING ********************************************
 *** The KEBA Kemro K2 System including software is not intended for safety control tasks! ***
 ***                       For further information see Comment tab!                        ***
 *********************************************************************************************)

IF evStartedStoppedData.MoveId = cMoldHeightAutomatic AND evStartedStoppedData.DeviceId = sv_DeviceId THEN
   IF evStartedStoppedData.State = nStopped OR evStartedStoppedData.State = nStartNotAllowed THEN
      //reset flag when movement in state nStopped OR nStartNotAllowed
      //we can not use a POSTUPDATE on sv_bDeviceReady and check for TRUE because the movement might be locked
      // -> sv_bDeviceReady never goes FALSE -> no POSTUPDATE is executed
      //also we can not use evMovementState because this one is not set by mold height adjust admin
      sv_bMoldHeightAutoAdjHMI := FALSE;
   END_IF;
END_IF;

;#END_EDIT_BLOCK END_ALGORITHM

END_ALGORITHM_BLOCK

#END_OF_IEC_PART

@Puma @IecEditor 6 114 @Pou 25
@@@BEG_Comment@@@
@h    ! WARNING !
@h    The Kemro K2 system (including software) only meets category B according to EN 954-1,
@h    thus it is not intended for usage in safety-relevant control applications in the field
@h    of personal safety (e.g. emergency stop).
@h    To implement potentially necessary safety-relevant control tasks, always use additional
@h    external safety devices that are intended for the particular purpose, and meet the necessary
@h    functional safety.
@h    For further information see EN 954-1 (EN ISO 13849-1) and/or the K2-x00 user manual, chapter
@h    "CE conformity, directives and standards".

This algo block starts the automatic mold height adjustment by calling the
system.FBManualButton with the correct parameters corresponding to a pressed Panel Button.
@@@END_Comment@@@

@BEG_Contents

@BEG_Func
@RT(17)FuncTreeContainer
1
@Var @RT(9)SET_ALARM @RT(0) @T @T @DERIVED 0 @F @RT(23)KEBA_STANDARD_PROCEDURE @F
@T
@BEG_Attrib
0 @RT(0) @RT(0)
@END_Attrib
1 1 @F @F @F @F

@END_Func

@BEG_Const
@RT(18)ConstTreeContainer
3
@Var @RT(6)nSetup @RT(0) @T @T @DERIVED 0 @F @RT(15)tnOperationMode @F
@T
@BEG_Attrib
0 @RT(1)0 @RT(36)Setup mode only for service engineer
@END_Attrib
1 1 @F @F @F @F

@Var @RT(9)cCompMold @RT(0) @T @F @DT @RT(4)DINT @RT(0) @T @T @BASIC 0 @F
@F @F
@T
@BEG_Attrib
0 @RT(3)101 @RT(14)Component Mold
@END_Attrib
1 1 @F @F @F @F

@Var @RT(15)cCompMoldHeight @RT(0) @T @F @DT @RT(4)DINT @RT(0) @T @T @BASIC 0 @F
@F @F
@T
@BEG_Attrib
0 @RT(3)124 @RT(21)Component Mold Height
@END_Attrib
1 1 @F @F @F @F

@END_Const

@BEG_Export

@BEG_Kind
@ALGORITHM_BLOCK @RT(14)ABManualButton @STRUCTURED_TEXT
@RT(0) @RT(0) @RT(0)
@END_Kind

@BEG_Dcl
@RT(16)DclTreeContainer
22
@Var @RT(9)PU_Task_7 @RT(0) @T @F @DT @RT(4)TASK @RT(0) @T @T @BASIC 0 @F
@F @F
@T
@BEG_Attrib
3 @RT(0) @RT(0) @RT(0)
@END_Attrib
1 7 @F @F @F @F

@Var @RT(9)EV_Task_7 @RT(0) @T @F @DT @RT(4)TASK @RT(0) @T @T @BASIC 0 @F
@F @F
@T
@BEG_Attrib
3 @RT(0) @RT(0) @RT(0)
@END_Attrib
1 7 @F @F @F @F

@Var @RT(28)erSetupModeRequiredForAdjust @RT(0) @T @F @DT @RT(5)ALARM @RT(0) @T @T @BASIC 0 @F
@F @F
@T
@BEG_Attrib
3 @RT(0) @RT(0) @RT(0)
@END_Attrib
1 7 @F @F @F @F

@Var @RT(16)evStartedStopped @RT(0) @T @T @DERIVED 0 @T @T @DT @RT(17)tevStartedStopped @RT(0) @T @T @UNKNOWN 0 @F
@F @F
@T
@BEG_Attrib
3 @RT(0) @RT(0) @RT(0)
@END_Attrib
1 7 @F @F @F @F

@Var @RT(21)sv_MoveMoldHeightAuto @RT(0) @T @T @DERIVED 0 @T @T @DT @RT(10)tsMoveData @RT(0) @T @T @UNKNOWN 0 @F
@F @F
@T
@BEG_Attrib
3 @RT(0) @RT(0) @RT(0)
@END_Attrib
1 8 @F @F @F @F

@Var @RT(30)sv_bAutoMoldHeightAdjustActive @RT(0) @T @F @DT @RT(4)BOOL @RT(0) @T @T @BASIC 0 @F
@F @F
@T
@BEG_Attrib
3 @RT(0) @RT(46)is TRUE when auto mold height adjust is acitve @RT(0)
@END_Attrib
1 8 @F @F @F @F

@Var @RT(25)sv_bLedAutoAdjust_ledAttr @RT(0) @T @F @DT @RT(4)BYTE @RT(0) @T @T @BASIC 0 @F
@F @F
@T
@BEG_Attrib
3 @RT(0) @RT(13)LED Attribute @RT(0)
@END_Attrib
1 8 @F @F @F @F

@Var @RT(20)sv_bHMILedAutoAdjust @RT(0) @T @F @DT @RT(4)BOOL @RT(0) @T @T @BASIC 0 @F
@F @F
@T
@BEG_Attrib
3 @RT(0) @RT(0) @RT(0)
@END_Attrib
1 8 @F @F @F @F

@Var @RT(28)sv_bHMILedAutoAdjust_ledAttr @RT(0) @T @F @DT @RT(4)BYTE @RT(0) @T @T @BASIC 0 @F
@F @F
@T
@BEG_Attrib
3 @RT(0) @RT(13)LED Attribute @RT(0)
@END_Attrib
1 8 @F @F @F @F

@Var @RT(17)sv_bLedAutoAdjust @RT(0) @T @F @DT @RT(4)BOOL @RT(0) @T @T @BASIC 0 @F
@F @F
@T
@BEG_Attrib
3 @RT(0) @RT(0) @RT(0)
@END_Attrib
1 8 @F @F @F @F

@Var @RT(13)sv_bInitStart @RT(0) @T @F @DT @RT(4)BOOL @RT(0) @T @T @BASIC 0 @F
@F @F
@T
@BEG_Attrib
3 @RT(0) @RT(0) @RT(0)
@END_Attrib
1 8 @F @F @F @F

@Var @RT(16)sv_OperationMode @RT(0) @T @T @DERIVED 0 @T @T @DT @RT(15)tnOperationMode @RT(0) @T @T @UNKNOWN 0 @F
@F @F
@T
@BEG_Attrib
3 @RT(0) @RT(0) @RT(0)
@END_Attrib
1 8 @F @F @F @F

@Var @RT(12)sv_bInitDone @RT(0) @T @F @DT @RT(4)BOOL @RT(0) @T @T @BASIC 0 @F
@F @F
@T
@BEG_Attrib
3 @RT(0) @RT(0) @RT(0)
@END_Attrib
1 8 @F @F @F @F

@Var @RT(11)sv_DeviceId @RT(0) @T @T @DERIVED 0 @T @T @DT @RT(10)tsDeviceId @RT(0) @T @T @UNKNOWN 0 @F
@F @F
@T
@BEG_Attrib
3 @RT(0) @RT(0) @RT(0)
@END_Attrib
1 8 @F @F @F @F

@Var @RT(24)sv_bMoldHeightAutoAdjHMI @RT(0) @T @F @DT @RT(4)BOOL @RT(0) @T @T @BASIC 0 @F
@F @F
@T
@BEG_Attrib
3 @RT(0) @RT(45)hmi can start/stop automh adjust with this SV @RT(0)
@END_Attrib
1 8 @F @F @F @F

@Var @RT(15)sv_bDeviceReady @RT(0) @T @F @DT @RT(4)BOOL @RT(0) @T @T @BASIC 0 @F
@F @F
@T
@BEG_Attrib
3 @RT(0) @RT(0) @RT(0)
@END_Attrib
1 8 @F @F @F @F

@Var @RT(14)fbManualButton @RT(0) @T @T @DERIVED 0 @T @T @DT @RT(18)FBManualButtonKeep @RT(0) @T @T @UNKNOWN 0 @F
@F @F
@T
@BEG_Attrib
3 @RT(0) @RT(0) @RT(0)
@END_Attrib
1 0 @F @F @F @F

@Var @RT(12)mpbMoldReady @RT(0) @T @T @REFTO 0 @T @DT @RT(4)BOOL @RT(0) @T @T @BASIC 0 @F
@F @F
@T
@BEG_Attrib
3 @RT(0) @RT(0) @RT(0)
@END_Attrib
1 0 @F @F @F @F

@Var @RT(18)mpbMoldHeightReady @RT(0) @T @T @REFTO 0 @T @DT @RT(4)BOOL @RT(0) @T @T @BASIC 0 @F
@F @F
@T
@BEG_Attrib
3 @RT(0) @RT(0) @RT(0)
@END_Attrib
1 0 @F @F @F @F

@Var @RT(10)g_b2Platen @RT(0) @T @F @DT @RT(4)BOOL @RT(0) @T @T @BASIC 0 @F
@F @F
@T
@BEG_Attrib
3 @RT(0) @RT(0) @RT(0)
@END_Attrib
1 6 @F @F @F @F

@Var @RT(11)mpbNutsOpen @RT(0) @T @T @REFTO 0 @T @DT @RT(4)BOOL @RT(0) @T @T @BASIC 0 @F
@F @F
@T
@BEG_Attrib
3 @RT(0) @RT(0) @RT(0)
@END_Attrib
1 0 @F @F @F @F

@Var @RT(17)mAlarmNutsNotOpen @RT(0) @T @T @DERIVED 0 @F @RT(7)tsAlarm @F
@T
@BEG_Attrib
3 @RT(0) @RT(0) @RT(0)
@END_Attrib
1 0 @F @F @F @F

@END_Dcl

@END_Export

@BEG_Body

6

@BEG_Export

@BEG_Algo
@ALGORITHM @RT(10)aStartStop @STRUCTURED_TEXT
@RT(0) @RT(0) @RT(0) @F @F
@END_Algo

@BEG_Dcl
@RT(16)DclTreeContainer
1
@Var @RT(6)bStart @RT(0) @T @F @DT @RT(4)BOOL @RT(0) @T @T @BASIC 0 @F
@F @F
@T
@BEG_Attrib
3 @RT(0) @RT(0) @RT(0)
@END_Attrib
1 1 @F @F @F @F

@END_Dcl

@END_Export

@BEG_Export

@BEG_Algo
@ALGORITHM @RT(12)aButtonStart @STRUCTURED_TEXT
@RT(0) @RT(0) @RT(0) @F @F
@END_Algo

@BEG_Dcl
@RT(16)DclTreeContainer
1
@Var @RT(12)bButtonStart @RT(0) @T @F @DT @RT(4)BOOL @RT(0) @T @T @BASIC 0 @F
@F @F
@T
@BEG_Attrib
3 @RT(0) @RT(0) @RT(0)
@END_Attrib
1 1 @F @F @F @F

@END_Dcl

@END_Export

@BEG_Export

@BEG_Algo
@POSTUPDATE_ALGORITHM @RT(9)pHMIStart @STRUCTURED_TEXT
@RT(0) @RT(24)sv_bMoldHeightAutoAdjHMI @RT(9)PU_Task_7 @F @F
@END_Algo

@BEG_Dcl
@RT(16)DclTreeContainer
0
@END_Dcl

@END_Export

@BEG_Export

@BEG_Algo
@POSTUPDATE_ALGORITHM @RT(11)pLedControl @STRUCTURED_TEXT
@RT(0) @RT(44)sv_bAutoMoldHeightAdjustActive,sv_bInitStart @RT(9)PU_Task_7 @F @F
@END_Algo

@BEG_Dcl
@RT(16)DclTreeContainer
2
@Var @RT(9)bInitDone @RT(0) @T @F @DT @RT(4)BOOL @RT(0) @T @T @BASIC 0 @F
@F @F
@T
@BEG_Attrib
3 @RT(0) @RT(0) @RT(0)
@END_Attrib
1 0 @F @F @F @F

@Var @RT(21)mbLedAutoAdjustExists @RT(0) @T @F @DT @RT(4)BOOL @RT(0) @T @T @BASIC 0 @F
@F @F
@T
@BEG_Attrib
3 @RT(5)FALSE @RT(0) @RT(0)
@END_Attrib
1 0 @F @F @F @F

@END_Dcl

@END_Export

@BEG_Export

@BEG_Algo
@POSTUPDATE_ALGORITHM @RT(9)pInitDone @STRUCTURED_TEXT
@RT(0) @RT(12)sv_bInitDone @RT(13)PU_Task_7(10) @F @F
@END_Algo

@BEG_Dcl
@RT(16)DclTreeContainer
3
@Var @RT(12)fbCheckReady @RT(0) @T @T @DERIVED 0 @T @T @DT @RT(12)FBCheckReady @RT(0) @T @T @UNKNOWN 0 @F
@F @F
@T
@BEG_Attrib
3 @RT(0) @RT(0) @RT(0)
@END_Attrib
1 0 @F @F @F @F

@Var @RT(8)DeviceId @RT(0) @T @T @DERIVED 0 @T @T @DT @RT(10)tsDeviceId @RT(0) @T @T @UNKNOWN 0 @F
@F @F
@T
@BEG_Attrib
3 @RT(0) @RT(0) @RT(0)
@END_Attrib
1 0 @F @F @F @F

@Var @RT(17)fbCheckPosReached @RT(0) @T @T @DERIVED 0 @F @RT(17)FBCheckPosReached @F
@T
@BEG_Attrib
3 @RT(0) @RT(0) @RT(0)
@END_Attrib
1 0 @F @F @F @F

@END_Dcl

@END_Export

@BEG_Export

@BEG_Algo
@EVENT_ALGORITHM @RT(17)evaStartedStopped @STRUCTURED_TEXT
@RT(0) @RT(16)evStartedStopped @RT(9)EV_Task_7 @F @F
@END_Algo

@BEG_Dcl
@RT(16)DclTreeContainer
1
@Var @RT(20)evStartedStoppedData @RT(0) @T @T @DERIVED 0 @T @T @DT @RT(21)tevStartedStoppedData @RT(0) @T @T @UNKNOWN 0 @F
@F @F
@T
@BEG_Attrib
3 @RT(0) @RT(0) @RT(0)
@END_Attrib
1 1 @F @F @F @F

@END_Dcl

@END_Export

@BEG_Body
@TL(37)
(**************************************** WARNING ********************************************
 *** The KEBA Kemro K2 System including software is not intended for safety control tasks! ***
 ***                       For further information see Comment tab!                        ***
 *********************************************************************************************)

IF (bStart AND (sv_OperationMode <> nSetup)) THEN
   //ignore button if operation mode is not setup
   SET_ALARM(Name := erSetupModeRequiredForAdjust,
            SubID1 := sv_DeviceId.CompId);
   sv_bMoldHeightAutoAdjHMI := FALSE;
   RETURN;
END_IF;

IF bStart AND g_b2Platen THEN
   //ignore button if lock nuts are not open
   IF NOT mpbNutsOpen^ THEN
      SET_ALARM(Name := mAlarmNutsNotOpen.AlarmId);
      sv_bMoldHeightAutoAdjHMI := FALSE;
      RETURN;
   END_IF;
END_IF;

IF (bStart AND sv_bDeviceReady) THEN
   IF (mpbMoldReady <> EMPTY AND NOT mpbMoldReady^) OR (mpbMoldHeightReady <> EMPTY AND NOT mpbMoldHeightReady^) THEN
      // auto adjust should be started and mold movement or mold adjust movement acitve
      // -> ignore manual button
      RETURN;
   END_IF;
END_IF;

(*@ MoldHeightAdjustN.ABManualButton.pButtonStart.Call the fbManualButton using the sv_MoveMoldHeightAuto parameters *)
IF (bStart AND sv_bDeviceReady) OR ((NOT bStart) AND (NOT sv_bDeviceReady)) THEN
   fbManualButton(bButton := TRUE, MoveId := sv_MoveMoldHeightAuto.MoveId, MoveDir := sv_MoveMoldHeightAuto.MoveDir);
END_IF;

@END_Body

@@@BEG_Comment@@@
@TL(3)
This algo starts the mold height automatic adjustment by calling the
system.FBManualButton with the correct parameters when the di_ButtonIn is
pressed. (post update).
@@@END_Comment@@@

@BEG_Body
@TL(9)
(**************************************** WARNING ********************************************
 *** The KEBA Kemro K2 System including software is not intended for safety control tasks! ***
 ***                       For further information see Comment tab!                        ***
 *********************************************************************************************)

IF bButtonStart THEN
    sv_bMoldHeightAutoAdjHMI := NOT sv_bMoldHeightAutoAdjHMI;
END_IF;

@END_Body

@@@BEG_Comment@@@
@TL(3)
This algo starts the mold height automatic adjustment by calling the
system.FBManualButton with the correct parameters when the di_ButtonIn is
pressed. (post update).
@@@END_Comment@@@

@BEG_Body
@TL(12)
(**************************************** WARNING ********************************************
 *** The KEBA Kemro K2 System including software is not intended for safety control tasks! ***
 ***                       For further information see Comment tab!                        ***
 *********************************************************************************************)

IF (sv_bMoldHeightAutoAdjHMI AND sv_bDeviceReady) THEN
    aStartStop(TRUE);
ELSIF ((NOT sv_bMoldHeightAutoAdjHMI) AND (NOT sv_bDeviceReady)) THEN
    aStartStop(FALSE);
END_IF;

@END_Body

@@@BEG_Comment@@@
@TL(3)
This algo starts the mold height automatic adjustment by calling the
system.FBManualButton with the correct parameters when the di_ButtonIn is
pressed. (post update).
@@@END_Comment@@@

@BEG_Body
@TL(22)
(**************************************** WARNING ********************************************
 *** The KEBA Kemro K2 System including software is not intended for safety control tasks! ***
 ***                       For further information see Comment tab!                        ***
 *********************************************************************************************)

IF NOT bInitDone THEN
    sv_bHMILedAutoAdjust_ledAttr := 16#3;
    IF IS_LINKED(sv_bLedAutoAdjust) AND IS_LINKED(sv_bLedAutoAdjust_ledAttr) THEN
        sv_bLedAutoAdjust_ledAttr := sv_bHMILedAutoAdjust_ledAttr;
        mbLedAutoAdjustExists := TRUE;
    ELSE
        mbLedAutoAdjustExists := FALSE;
    END_IF;

    bInitDone := TRUE;
END_IF;

sv_bHMILedAutoAdjust := sv_bAutoMoldHeightAdjustActive;
IF mbLedAutoAdjustExists THEN
    sv_bLedAutoAdjust := sv_bHMILedAutoAdjust;
END_IF;

@END_Body

@@@BEG_Comment@@@
@TL(0)

@@@END_Comment@@@

@BEG_Body
@TL(29)
(**************************************** WARNING ********************************************
 *** The KEBA Kemro K2 System including software is not intended for safety control tasks! ***
 ***                       For further information see Comment tab!                        ***
 *********************************************************************************************)

//get reference to ready flag of mold function unit
DeviceId.CompId := cCompMold;
DeviceId.IndexId := sv_DeviceId.IndexId;
fbCheckReady(DeviceId := DeviceId);
mpbMoldReady := fbCheckReady.pbReady;

//get reference to ready flag of mold adjust function unit
DeviceId.CompId := cCompMoldHeight;
DeviceId.IndexId := sv_DeviceId.IndexId;
fbCheckReady(DeviceId := DeviceId);
mpbMoldHeightReady := fbCheckReady.pbReady;

//get reference to mold nut open movement and save according alarm
IF g_b2Platen THEN
   DeviceId.CompId := cCompMoldNuts;
   DeviceId.IndexId := sv_DeviceId.IndexId;
   fbCheckPosReached(DeviceId := DeviceId,
                     MoveDir := cMoveOpen,
                     MoveId := cMoveOpen);

   mpbNutsOpen := fbCheckPosReached.pbPosReached;
   mAlarmNutsNotOpen := fbCheckPosReached.Alarm;
END_IF;

@END_Body

@@@BEG_Comment@@@
@TL(0)

@@@END_Comment@@@

@BEG_Body
@TL(18)
(**************************************** WARNING ********************************************
 *** The KEBA Kemro K2 System including software is not intended for safety control tasks! ***
 ***                       For further information see Comment tab!                        ***
 *********************************************************************************************)

IF evStartedStoppedData.MoveId = cMoldHeightAutomatic AND evStartedStoppedData.DeviceId = sv_DeviceId THEN
   IF evStartedStoppedData.State = nStopped OR evStartedStoppedData.State = nStartNotAllowed THEN
      //reset flag when movement in state nStopped OR nStartNotAllowed
      //we can not use a POSTUPDATE on sv_bDeviceReady and check for TRUE because the movement might be locked
      // -> sv_bDeviceReady never goes FALSE -> no POSTUPDATE is executed
      //also we can not use evMovementState because this one is not set by mold height adjust admin
      sv_bMoldHeightAutoAdjHMI := FALSE;
   END_IF;
END_IF;

@END_Body

@@@BEG_Comment@@@
@TL(2)
Manage list and count of currently started movments
in sv_StartedMovements when receiving evStartedStopped events
@@@END_Comment@@@
@END_Body

@END_Contents

(* ---- ABMeasure.pu ---- *)
(*
@h    ! WARNING !
@h    The Kemro K2 system (including software) only meets category B according to EN 954-1,
@h    thus it is not intended for usage in safety-relevant control applications in the field
@h    of personal safety (e.g. emergency stop).
@h    To implement potentially necessary safety-relevant control tasks, always use additional
@h    external safety devices that are intended for the particular purpose, and meet the necessary
@h    functional safety.
@h    For further information see EN 954-1 (EN ISO 13849-1) and/or the K2-x00 user manual, chapter
@h    "CE conformity, directives and standards".

This algorithm block is used for measuring the mold height position.
*)

IMPORT_OVER_LISTFILE
 tsMoldHeightPositions

END_IMPORT

ALGORITHM_BLOCK ABMeasure #DUMMY_EDIT_BLOCK

SYSTEM_VAR
 sv_rDistancePerImpulse : REAL;
 sv_iAbsoluteImpulsesFromOrigin : DINT;
 sv_MoldHeightPositions : tsMoldHeightPositions;
 sv_rActMoldHeightPosition : REAL;
 sv_bInitDone : BOOL;
END_VAR

SYSTEM_OBJECT
 TaskAnalog : TASK;
 PU_Task_7 : TASK;
END_OBJECT

VAR_EXTERNAL
 g_b2Platen : BOOL;
 g_bDirectLock : BOOL;
END_VAR

(*
The measurement of mold height position works by converting the
counted impulses of mold hieght movement (counted by MoldHeightN.ABMeasure.paMeasure)
into a position using a factor (which is calculated while calibrating the impulse-distance-relationship)
*)

PROCESS_ALGORITHM paMeasurePosition ON TaskAnalog(1000)

#BEGIN_EDIT_BLOCK
(**************************************** WARNING ********************************************
 *** The KEBA Kemro K2 System including software is not intended for safety control tasks! ***
 ***                       For further information see Comment tab!                        ***
 *********************************************************************************************)

sv_rActMoldHeightPosition := sv_MoldHeightPositions.rOriginMoldHeightPosition + (DINT_TO_REAL(sv_iAbsoluteImpulsesFromOrigin) * sv_rDistancePerImpulse);

;#END_EDIT_BLOCK END_ALGORITHM

POSTUPDATE_ALGORITHM pInitDone ON PU_Task_7 WITH sv_bInitDone

#BEGIN_EDIT_BLOCK
(**************************************** WARNING ********************************************
 *** The KEBA Kemro K2 System including software is not intended for safety control tasks! ***
 ***                       For further information see Comment tab!                        ***
 *********************************************************************************************)

IF NOT g_b2Platen AND NOT g_bDirectLock THEN
   START_PROCESS_ALGORITHM(paMeasurePosition);
END_IF;

;#END_EDIT_BLOCK END_ALGORITHM

END_ALGORITHM_BLOCK

#END_OF_IEC_PART

@Puma @IecEditor 6 22 @Pou 25
@@@BEG_Comment@@@
@h    ! WARNING !
@h    The Kemro K2 system (including software) only meets category B according to EN 954-1,
@h    thus it is not intended for usage in safety-relevant control applications in the field
@h    of personal safety (e.g. emergency stop).
@h    To implement potentially necessary safety-relevant control tasks, always use additional
@h    external safety devices that are intended for the particular purpose, and meet the necessary
@h    functional safety.
@h    For further information see EN 954-1 (EN ISO 13849-1) and/or the K2-x00 user manual, chapter
@h    "CE conformity, directives and standards".

This algorithm block is used for measuring the mold height position.
@@@END_Comment@@@

@BEG_Contents

@BEG_Func
@RT(17)FuncTreeContainer
0
@END_Func

@BEG_Const
@RT(18)ConstTreeContainer
0
@END_Const

@BEG_Export

@BEG_Kind
@ALGORITHM_BLOCK @RT(9)ABMeasure @STRUCTURED_TEXT
@RT(0) @RT(0) @RT(0)
@END_Kind

@BEG_Dcl
@RT(16)DclTreeContainer
9
@Var @RT(10)TaskAnalog @RT(0) @T @T @RENAMED 0 @T @T @DT @RT(4)TASK @RT(0) @T @T @BASIC 0 @F
@F @F
@T
@BEG_Attrib
3 @RT(0) @RT(0) @RT(0)
@END_Attrib
1 7 @F @F @F @F

@Var @RT(22)sv_rDistancePerImpulse @RT(0) @T @F @DT @RT(4)REAL @RT(0) @T @T @BASIC 0 @F
@F @F
@T
@BEG_Attrib
3 @RT(0) @RT(0) @RT(0)
@END_Attrib
1 8 @F @F @F @F

@Var @RT(30)sv_iAbsoluteImpulsesFromOrigin @RT(0) @T @F @DT @RT(4)DINT @RT(0) @T @T @BASIC 0 @F
@F @F
@T
@BEG_Attrib
3 @RT(0) @RT(0) @RT(0)
@END_Attrib
1 8 @F @F @F @F

@Var @RT(22)sv_MoldHeightPositions @RT(0) @T @T @DERIVED 0 @F @RT(21)tsMoldHeightPositions @F
@T
@BEG_Attrib
3 @RT(0) @RT(0) @RT(0)
@END_Attrib
1 8 @F @F @F @F

@Var @RT(25)sv_rActMoldHeightPosition @RT(0) @T @F @DT @RT(4)REAL @RT(0) @T @T @BASIC 0 @F
@F @F
@T
@BEG_Attrib
3 @RT(0) @RT(0) @RT(0)
@END_Attrib
1 8 @F @F @F @F

@Var @RT(9)PU_Task_7 @RT(0) @T @T @RENAMED 0 @T @T @DT @RT(4)TASK @RT(0) @T @T @BASIC 0 @F
@F @F
@T
@BEG_Attrib
3 @RT(0) @RT(0) @RT(0)
@END_Attrib
1 7 @F @F @F @F

@Var @RT(12)sv_bInitDone @RT(0) @T @T @RENAMED 0 @T @T @DT @RT(4)BOOL @RT(0) @T @T @BASIC 0 @F
@F @F
@T
@BEG_Attrib
3 @RT(0) @RT(0) @RT(0)
@END_Attrib
1 8 @F @F @F @F

@Var @RT(10)g_b2Platen @RT(0) @T @F @DT @RT(4)BOOL @RT(0) @T @T @BASIC 0 @F
@F @F
@T
@BEG_Attrib
3 @RT(0) @RT(0) @RT(0)
@END_Attrib
1 6 @F @F @F @F

@Var @RT(13)g_bDirectLock @RT(0) @T @F @DT @RT(4)BOOL @RT(0) @T @T @BASIC 0 @F
@F @F
@T
@BEG_Attrib
3 @RT(0) @RT(0) @RT(0)
@END_Attrib
1 6 @F @F @F @F

@END_Dcl

@END_Export

@BEG_Body

2

@BEG_Export

@BEG_Algo
@PROCESS_ALGORITHM @RT(17)paMeasurePosition @STRUCTURED_TEXT
@RT(0) @RT(0) @RT(16)TaskAnalog(1000) @F @F
@END_Algo

@BEG_Dcl
@RT(16)DclTreeContainer
0
@END_Dcl

@END_Export

@BEG_Export

@BEG_Algo
@POSTUPDATE_ALGORITHM @RT(9)pInitDone @STRUCTURED_TEXT
@RT(0) @RT(12)sv_bInitDone @RT(9)PU_Task_7 @F @F
@END_Algo

@BEG_Dcl
@RT(16)DclTreeContainer
0
@END_Dcl

@END_Export

@BEG_Body
@TL(7)
(**************************************** WARNING ********************************************
 *** The KEBA Kemro K2 System including software is not intended for safety control tasks! ***
 ***                       For further information see Comment tab!                        ***
 *********************************************************************************************)

sv_rActMoldHeightPosition := sv_MoldHeightPositions.rOriginMoldHeightPosition + (DINT_TO_REAL(sv_iAbsoluteImpulsesFromOrigin) * sv_rDistancePerImpulse);

@END_Body

@@@BEG_Comment@@@
@TL(3)
The measurement of mold height position works by converting the
counted impulses of mold hieght movement (counted by MoldHeightN.ABMeasure.paMeasure)
into a position using a factor (which is calculated while calibrating the impulse-distance-relationship)
@@@END_Comment@@@

@BEG_Body
@TL(9)
(**************************************** WARNING ********************************************
 *** The KEBA Kemro K2 System including software is not intended for safety control tasks! ***
 ***                       For further information see Comment tab!                        ***
 *********************************************************************************************)

IF NOT g_b2Platen AND NOT g_bDirectLock THEN
   START_PROCESS_ALGORITHM(paMeasurePosition);
END_IF;

@END_Body

@@@BEG_Comment@@@
@TL(0)

@@@END_Comment@@@
@END_Body

@END_Contents
